KUKA KRL program: reinigung.src, reinigung.dat

--- reinigung.src ---
&ACCESS RVO1
&REL 42
&COMMENT dai_cleaning
&USER PKL_AST
&PARAM DISKPATH = KRC:\R1\H_Prog
&PARAM version = 0.1
DEF reinigung( )
;FOLD INI
  ;FOLD BASISTECH INI
    GLOBAL INTERRUPT DECL 3 WHEN $STOPMESS==TRUE DO IR_STOPM ( )
    BAS (#INITMOV,0 )
  ;ENDFOLD (BASISTECH INI)
;FOLD SPOTTECH INI
USERSPOT(#INIT)
;ENDFOLD (SPOTTECH INI)
;FOLD GRIPPERTECH INI
USER_GRP(0,DUMMY,DUMMY,GDEFAULT)
;ENDFOLD (GRIPPERTECH INI)
;FOLD USER INI

;Make your modifications here
;FOLD COLLISION_V_3.01 INI ;%{E}
    IF (COLLISION_DATA[1].I_NR>0) THEN
    GLOBAL INTERRUPT DECL 21 WHEN $IN[COLLISION_DATA[1].I_NR]==FALSE DO COLLSTOP (1,0 )
    ENDIF
    IF (COLLISION_DATA[2].I_NR>0) THEN
    GLOBAL INTERRUPT DECL 22 WHEN $IN[COLLISION_DATA[2].I_NR]==FALSE DO COLLSTOP (2,0 )
    ENDIF
    IF (COLLISION_DATA[3].I_NR>0) THEN
    GLOBAL INTERRUPT DECL 23 WHEN $IN[COLLISION_DATA[3].I_NR]==FALSE DO COLLSTOP (3,0 )
    ENDIF
    IF (COLLISION_DATA[4].I_NR>0) THEN
    GLOBAL INTERRUPT DECL 24 WHEN $IN[COLLISION_DATA[4].I_NR]==FALSE DO COLLSTOP (4,0 )
    ENDIF
;ENDFOLD (Collision)

;ENDFOLD (USER INI)

;ENDFOLD (INI)

; Caracterização dos meios de produção:
; Versão Atual:
; 08/06/2013 12:00 Name: P13.050-R1 CHANGES: Limpeza

chk_w8_wechs_ok ( )              ; CHECK TOOL CHANGE

if not nearE6Axis(XHOME5) then

	;FOLD PTP HOME Vel=100 % DEFAULT;%{PE}%R 5.5.24,%MKUKATPBASIS,%CMOVE,%VPTP,%P 1:PTP, 2:HOME, 3:, 5:100, 7:DEFAULT
	$BWDSTART=FALSE
	PDAT_ACT=PDEFAULT
	FDAT_ACT=FHOME
	BAS(#PTP_PARAMS,100)
	$H_POS=XHOME
	PTP XHOME
	;ENDFOLD

endif

$Axis_Home[5]=XHOME5

;FOLD ; Ponto de limpeza;%{PE}%R 8.2.20,%MKUKATPBASIS,%CCOMMENT,%VNORMAL,%P 2:Ponto  de  limpeza
;ENDFOLD
;FOLD PTP P2 Vel=100 % PDAT10 Tool[0] Base[0];%{PE}%R 8.2.20,%MKUKATPBASIS,%CMOVE,%VPTP,%P 1:PTP, 2:P2, 3:, 5:100, 7:PDAT10
$BWDSTART=FALSE
PDAT_ACT=PPDAT10
FDAT_ACT=FP2
BAS(#PTP_PARAMS,100)
PTP XP2
;ENDFOLD

MSG_SHOW("DAI_H_Prog",#notify,999,"dai_cleaning_0")
;FOLD OUT 3218 'WPER:Wartungspos. erreicht'  State= TRUE ;%{PE}%R 5.2.22,%MKUKATPBASIS,%COUT,%VOUTX,%P 2:3218, 3:WPER:Wartungspos. erreicht, 5:TRUE, 6:
    $OUT[3218]=TRUE
;ENDFOLD
Halt
;FOLD WAIT FOR ( NOT IN 3218 'ANFWP:Anforderung Wartungspos.' );%{PE}%R 5.2.22,%MKUKATPBASIS,%CEXT_WAIT_FOR,%VEXT_WAIT_FOR,%P 2:, 4:NOT, 5:$IN, 6:3218, 7:ANFWP:Anforderung Wartungspos., 9:
    WAIT FOR  (  NOT $IN[3218] )
;ENDFOLD
;FOLD OUT 3218 'WPER:Wartungspos. erreicht'  State= FALSE ;%{PE}%R 5.2.22,%MKUKATPBASIS,%COUT,%VOUTX,%P 2:3218, 3:WPER:Wartungspos. erreicht, 5:FALSE, 6:
    $OUT[3218]=FALSE
;ENDFOLD


;FOLD PTP HOME Vel=100 % DEFAULT;%{PE}%R 5.5.24,%MKUKATPBASIS,%CMOVE,%VPTP,%P 1:PTP, 2:HOME, 3:, 5:100, 7:DEFAULT
$BWDSTART=FALSE
PDAT_ACT=PDEFAULT
FDAT_ACT=FHOME
BAS(#PTP_PARAMS,100)
$H_POS=XHOME
PTP XHOME
;ENDFOLD
END

--- reinigung.dat ---
&ACCESS RVO1
&REL 42
&COMMENT dai_cleaning
&USER PKL_AST
&PARAM DISKPATH = KRC:\R1\H_Prog
&PARAM version = 0.1
DEFDAT  reinigung
;FOLD EXTERNAL DECLARATIONS;%{PE}%MKUKATPBASIS,%CEXT,%VCOMMON,%P
;FOLD GRIPPERTECH EXT
EXT  H50 (INT  :IN,INT  :IN,INT  :IN,GRP_TYP  :IN )
;ENDFOLD (GRIPPERTECH EXT)
;FOLD SPOTTECH EXT
EXT  USERSPOT (S_COMMAND  :IN,SPOT_TYPE  :IN )
;ENDFOLD (SPOTTECH EXT)
;FOLD BASISTECH EXT;%{PE}%MKUKATPBASIS,%CEXT,%VEXT,%P
EXT  BAS (BAS_COMMAND  :IN,REAL  :IN )
DECL INT SUCCESS
;ENDFOLD (BASISTECH EXT)
;FOLD USER EXT;%{E}%MKUKATPUSER,%CEXT,%VEXT,%P
;Make here your modifications
;FOLD COLLISION
EXT  COLLSTOP (INT  :IN,INT  :IN )
;ENDFOLD  (Collision)
;ENDFOLD (USER EXT)
;ENDFOLD (EXTERNAL DECLERATIONS)

DECL BASIS_SUGG_T LAST_BASIS={POINT1[] "P3                      ",POINT2[] "P3                      ",CP_PARAMS[] "CPDAT0                  ",PTP_PARAMS[] "PDAT11                  ",CONT[] "C_DIS                   ",CP_VEL[] "2.0                     ",PTP_VEL[] "100                     ",SYNC_PARAMS[] "SYNCDAT                 ",SPL_NAME[] "S0                      "}





DECL E6POS XP2={X 135.209396,Y 1363.53198,Z 1543.15002,A 2.14462209,B -35.68787,C -90.0461731,S 6,T 19,E1 -419.038788,E2 0.0,E3 0.0,E4 0.0,E5 0.0,E6 0.0}
DECL FDAT FP2={TOOL_NO 0,BASE_NO 0,IPO_FRAME #BASE,POINT2[] " ",TQ_STATE FALSE}
DECL PDAT PPDAT10={VEL 100.0,ACC 100.0,APO_DIST 100.0,APO_MODE #CDIS}
ENDDAT
